# B&R Automation Studio project SuperTrak_Distribution (part 3)

#### ReadErrorMessages.st - Read error messages task
```iecst
(*********************************************************************************
 * Copyright: Bernecker + Rainer
 * Author:  B+R
 * Created:  June 30, 2017/08:15 AM
 *********************************************************************************
 *********************************************************************************
 * Version History:
 * -------------------------------------------------------------------------------
 * V 1.00.0   June 30, 2017/08:15 AM  First Version
 *********************************************************************************
 * Description:
 * -------------------------------------------------------------------------------
 * June 30, 2017/08:15 AM AM V1.00.0:
 * This task is used for Error handling
 * Error number are read from the FUB and converted to messages
 * This messages are used for the visualization
 *********************************************************************************)

ACTION ReadErrorMessages:

	brsmemset(ADR(ErrorInfo),0,SIZEOF(ErrorInfo));

	IF EDGENEG(AcknowledgeAll) THEN
		StControl_0.ErrorReset										:= FALSE;
		FOR Index := 0 TO (SIZEOF(StSection_) / SIZEOF(StSection_[0])) - 1 DO
			StSection_[Index].ErrorReset							:= FALSE;
		END_FOR;
		FOR Index := 0 TO (SIZEOF(StTargetExt_) / SIZEOF(StTargetExt_[0])) - 1 DO
			StTargetExt_[Index].ErrorReset							:= FALSE;
		END_FOR;
		StWritePnu_Region.ErrorReset								:= FALSE;
		StReadPnu_Region.ErrorReset									:= FALSE;
	END_IF;

	FOR Index := 0 TO (SIZEOF(StSection_) / SIZEOF(StSection_[0])) - 1 DO
		////////////////////////////////////////////////////////////
		////////////////////////////////////////////////////////////
		//Check if fault is active to output the correct error msg
		Counter		:= 0;
		FOR FaultBitCounter := 0 TO 31 DO
			IF BIT_TST(StSection_[Index].Info.SuperTrak.SectionFaultBits,FaultBitCounter) THEN
				// Set error
				FaultBit											:= FaultBitCounter;
				ErrorInfo.StSection[Index].ErrorText[Counter]		:= ErrorTexts[FaultBit];
				ErrorInfo.StSection[Index].Error[Counter]			:= FaultBit;
				Counter			:= Counter + 1;
			END_IF;
		END_FOR;

		IF StSection_[Index].StatusID <> stCOM_NO_ERROR THEN
			ErrorInfo.StSection[Index].StatusID				:= StSection_[Index].StatusID;

			// Get the needed text
			CASE ErrorInfo.StSection[Index].StatusID OF
				stCOM_ERR_FB_INSTANCE_REG:
					ErrorInfo.StSection[Index].ErrorText[Counter]:= 'Instance of this function block already registered';

				stCOM_ERR_WRONG_PARAMETER:
					ErrorInfo.StSection[Index].ErrorText[Counter]:= 'Wrong parameter';

				stCOM_ERR_COMMUNICAITON_TIME_OUT:
					ErrorInfo.StSection[Index].ErrorText[Counter]:= 'Timeout for communication to SuperTrak';

				stCOM_ERR_NO_STCONTROL_REG:
					ErrorInfo.StSection[Index].ErrorText[Counter]:= 'There is no instance of StControl registered';

				stCOM_ERR_WRONG_CONFIG:
					ErrorInfo.StSection[Index].ErrorText[Counter]:= 'Address not valid, or Target/Section/PalletID not vaild';

				stCOM_ERR_CMD_NOT_EXECUTED:
					ErrorInfo.StSection[Index].ErrorText[Counter]:= 'Command could not be executed successfully';

				stCOM_ERR_SERVICE_CHANNEL_FAULT:
					ErrorInfo.StSection[Index].ErrorText[Counter]:= 'SuperTrak responded with an error to a service channel request';

				stCOM_ERR_CMD_HANDSHAKE:
					ErrorInfo.StSection[Index].ErrorText[Counter]:= 'CommandComplete flag is true before command execution';

			END_CASE;
		END_IF;

		////////////////////////////////////////////////////////////
		////////////////////////////////////////////////////////////
		//Check if warning is active to output the correct error msg
		Counter		:= 0;
		FOR FaultBitCounter := 0 TO 31 DO
			IF BIT_TST(StSection_[Index].Info.SuperTrak.SectionWarningBits,FaultBitCounter) THEN
				// Set warning
				WarningBit											:= FaultBitCounter;
				ErrorInfo.StSection[Index].WarningText[Counter]		:= WarningTexts[WarningBit];
				ErrorInfo.StSection[Index].Warning[Counter]			:= WarningBit;
				Counter	:= Counter + 1;
			END_IF;
		END_FOR;

		IF StSection_[Index].StatusID <> stCOM_NO_ERROR THEN
			// Get the needed text
			CASE ErrorInfo.StSection[Index].StatusID OF
				stCOM_WRN_ENABLE_SIGNAL_SOURCE:
					ErrorInfo.StSection[Index].WarningText[Counter]:= 'Enable signal source configuration does not allow this command';

				stCOM_INFO_COMM_STRUCT_TOO_BIG:
					ErrorInfo.StSection[Index].WarningText[Counter]:= 'The communication structure is too big';

			END_CASE;
		END_IF;
	END_FOR;

	///////////////////////////////////////////////////////////
	///////////////////////////////////////////////////////////
	// Use the actual selected Section to display
	// Count up the section on the Temperatures Visu page
	IF EDGEPOS(CountUpAlarm) THEN
		VisuAlarmSection		:= VisuAlarmSection + 1;
		// Check for last section
		IF VisuAlarmSection = (MAX_SECTIONS+1) THEN
			VisuAlarmSection	:= 1;
		END_IF;
		CountUpAlarm			:= FALSE;
		// Count down the section on the Temperatures Visu page
	ELSIF EDGEPOS(CountDownAlarm) THEN
		VisuAlarmSection		:= VisuAlarmSection - 1;
		// Check for first section
		IF VisuAlarmSection = 0 THEN
			VisuAlarmSection	:= MAX_SECTIONS;
		END_IF;
		CountDownAlarm			:= FALSE;
	END_IF;

	VisuAlarmSectionText		:= ErrorInfo.StSection[VisuAlarmSection-1].ErrorText;
	VisuWarningSectionText		:= ErrorInfo.StSection[VisuAlarmSection-1].WarningText;

	IF AcknowledgeSelectedSection AND AcknowledgeAll = FALSE THEN
		StSection_[VisuAlarmSection-1].ErrorReset		:= TRUE;
	END_IF;

	///////////////////////////////////////////////////////////
	///////////////////////////////////////////////////////////
	// Check if fault is active to output the correct error msg
	Counter	:= 0;
	FOR Index := 0 TO (SIZEOF(StTargetExt_) / SIZEOF(StTargetExt_[0])) - 1 DO
		// Get the StatusID of the FUB
		IF StTargetExt_[Index].StatusID <> stCOM_NO_ERROR THEN
			ErrorInfo.StTargetExt.StatusID[Counter]			:= StTargetExt_[Index].StatusID;
			ErrorInfo.StTargetExt.TargetID[Counter]			:= Index + 1;

			// Get the needed text
			CASE ErrorInfo.StTargetExt.StatusID[Counter] OF
				stCOM_ERR_FB_INSTANCE_REG:
					ErrorInfo.StTargetExt.ErrorText[Counter]:= 'Instance of this function block already registered';

				stCOM_ERR_WRONG_PARAMETER:
					ErrorInfo.StTargetExt.ErrorText[Counter]:= 'Wrong parameter';

				stCOM_ERR_COMMUNICAITON_TIME_OUT:
					ErrorInfo.StTargetExt.ErrorText[Counter]:= 'Timeout for communication to SuperTrak';

				stCOM_ERR_NO_STCONTROL_REG:
					ErrorInfo.StTargetExt.ErrorText[Counter]:= 'There is no instance of StControl registered';

				stCOM_ERR_WRONG_CONFIG:
					ErrorInfo.StTargetExt.ErrorText[Counter]:= 'Address not valid, or Target/Section/PalletID not vaild';

				stCOM_ERR_CMD_NOT_EXECUTED:
					ErrorInfo.StTargetExt.ErrorText[Counter]:= 'Command could not be executed successfully';

				stCOM_ERR_SERVICE_CHANNEL_FAULT:
					ErrorInfo.StTargetExt.ErrorText[Counter]:= 'SuperTrak responded with an error to a service channel request';

				stCOM_ERR_CMD_HANDSHAKE:
					ErrorInfo.StTargetExt.ErrorText[Counter]:= 'CommandComplete flag is true before command execution';

				stCOM_WRN_ENABLE_SIGNAL_SOURCE:
					ErrorInfo.StTargetExt.ErrorText[Counter]:= 'Enable signal source configuration does not allow this command';

				stCOM_INFO_COMM_STRUCT_TOO_BIG:
					ErrorInfo.StTargetExt.ErrorText[Counter]:= 'The communication structure is too big';

			END_CASE;
			Counter	:= Counter + 1;
		END_IF;
	END_FOR;

	IF AcknowledgeSelectedTarget AND AcknowledgeAll = FALSE THEN
		IF (ErrorInfo.StTargetExt.TargetID[SelectedTarget] -1) >= 0 AND (ErrorInfo.StTargetExt.TargetID[SelectedTarget] -1) < 255 THEN
			StTargetExt_[ErrorInfo.StTargetExt.TargetID[SelectedTarget] -1].ErrorReset		:= TRUE;
		END_IF;
	ELSIF AcknowledgeAll = FALSE THEN
		IF (ErrorInfo.StTargetExt.TargetID[SelectedTarget] -1) >= 0 AND (ErrorInfo.StTargetExt.TargetID[SelectedTarget] -1) < 255 THEN
			StTargetExt_[ErrorInfo.StTargetExt.TargetID[SelectedTarget] -1].ErrorReset		:= FALSE;
		END_IF;
	END_IF;

	///////////////////////////////////////////////////////////
	///////////////////////////////////////////////////////////
	// Check if fault is active to output the correct error msg
	Counter	:= 0;
	FOR Index := 0 TO (SIZEOF(StPallet_) / SIZEOF(StPallet_[0])) - 1 DO
		// Get the StatusID of the FUB
		IF StPallet_[Index].StatusID <> stCOM_NO_ERROR THEN
			ErrorInfo.StPallet.StatusID[Counter]			:= StPallet_[Index].StatusID;
			ErrorInfo.StPallet.ShuttleID[Counter]			:= Index + 1;

			// Get the needed text
			CASE ErrorInfo.StPallet.StatusID[Counter] OF
				stCOM_ERR_FB_INSTANCE_REG:
					ErrorInfo.StPallet.ErrorText[Counter]:= 'Instance of this function block already registered';

				stCOM_ERR_WRONG_PARAMETER:
					ErrorInfo.StPallet.ErrorText[Counter]:= 'Wrong parameter';

				stCOM_ERR_COMMUNICAITON_TIME_OUT:
					ErrorInfo.StPallet.ErrorText[Counter]:= 'Timeout for communication to SuperTrak';

				stCOM_ERR_NO_STCONTROL_REG:
					ErrorInfo.StPallet.ErrorText[Counter]:= 'There is no instance of StControl registered';

				stCOM_ERR_WRONG_CONFIG:
					ErrorInfo.StPallet.ErrorText[Counter]:= 'Address not valid, or Target/Section/PalletID not vaild';

				stCOM_ERR_CMD_NOT_EXECUTED:
					ErrorInfo.StPallet.ErrorText[Counter]:= 'Command could not be executed successfully';

				stCOM_ERR_SERVICE_CHANNEL_FAULT:
					ErrorInfo.StPallet.ErrorText[Counter]:= 'SuperTrak responded with an error to a service channel request';

				stCOM_ERR_CMD_HANDSHAKE:
					ErrorInfo.StPallet.ErrorText[Counter]:= 'CommandComplete flag is true before command execution';

				stCOM_WRN_ENABLE_SIGNAL_SOURCE:
					ErrorInfo.StPallet.ErrorText[Counter]:= 'Enable signal source configuration does not allow this command';

				stCOM_INFO_COMM_STRUCT_TOO_BIG:
					ErrorInfo.StPallet.ErrorText[Counter]:= 'The communication structure is too big';

			END_CASE;
			Counter	:= Counter + 1;
		END_IF;
	END_FOR;

	IF AcknowledgeSelectedShuttle AND AcknowledgeAll = FALSE THEN
		IF (ErrorInfo.StPallet.ShuttleID[SelectedShuttle] -1) >= 0 AND (ErrorInfo.StPallet.ShuttleID[SelectedShuttle] -1) < 255 THEN
			StPallet_[ErrorInfo.StPallet.ShuttleID[SelectedShuttle] -1].ErrorReset		:= TRUE;
		END_IF;
	ELSIF AcknowledgeAll = FALSE THEN
		IF (ErrorInfo.StPallet.ShuttleID[SelectedShuttle] -1) >= 0 AND (ErrorInfo.StPallet.ShuttleID[SelectedShuttle] -1) < 255 THEN
			StPallet_[ErrorInfo.StPallet.ShuttleID[SelectedShuttle] -1].ErrorReset		:= FALSE;
		END_IF;
	END_IF;

	///////////////////////////////////////////////////////////
	///////////////////////////////////////////////////////////
	//Check if fault is active to output the correct error msg
	ErrorInfo.StReadPnu_Region.StatusID			:= StReadPnu_Region.StatusID;
	// Get the needed text
	CASE ErrorInfo.StReadPnu_Region.StatusID OF
		stCOM_ERR_FB_INSTANCE_REG:
			ErrorInfo.StReadPnu_Region.ErrorText:= 'Instance of this function block already registered';

		stCOM_ERR_WRONG_PARAMETER:
			ErrorInfo.StReadPnu_Region.ErrorText:= 'Wrong parameter';

		stCOM_ERR_COMMUNICAITON_TIME_OUT:
			ErrorInfo.StReadPnu_Region.ErrorText:= 'Timeout for communication to SuperTrak';

		stCOM_ERR_NO_STCONTROL_REG:
			ErrorInfo.StReadPnu_Region.ErrorText:= 'There is no instance of StControl registered';

		stCOM_ERR_WRONG_CONFIG:
			ErrorInfo.StReadPnu_Region.ErrorText:= 'Address not valid, or Target/Section/PalletID not vaild';

		stCOM_ERR_CMD_NOT_EXECUTED:
			ErrorInfo.StReadPnu_Region.ErrorText:= 'Command could not be executed successfully';

		stCOM_ERR_SERVICE_CHANNEL_FAULT:
			ErrorInfo.StReadPnu_Region.ErrorText:= 'SuperTrak responded with an error to a service channel request';

		stCOM_ERR_CMD_HANDSHAKE:
			ErrorInfo.StReadPnu_Region.ErrorText:= 'CommandComplete flag is true before command execution';

		stCOM_WRN_ENABLE_SIGNAL_SOURCE:
			ErrorInfo.StReadPnu_Region.ErrorText:= 'Enable signal source configuration does not allow this command';

		stCOM_INFO_COMM_STRUCT_TOO_BIG:
			ErrorInfo.StReadPnu_Region.ErrorText:= 'The communication structure is too big';

	END_CASE;

	///////////////////////////////////////////////////////////
	///////////////////////////////////////////////////////////
	//Check if fault is active to output the correct error msg
	ErrorInfo.StWritePnu_Region.StatusID		:= StWritePnu_Region.StatusID;
	// Get the needed text
	CASE ErrorInfo.StWritePnu_Region.StatusID OF
		stCOM_ERR_FB_INSTANCE_REG:
			ErrorInfo.StWritePnu_Region.ErrorText:= 'Instance of this function block already registered';

		stCOM_ERR_WRONG_PARAMETER:
			ErrorInfo.StWritePnu_Region.ErrorText:= 'Wrong parameter';

		stCOM_ERR_COMMUNICAITON_TIME_OUT:
			ErrorInfo.StWritePnu_Region.ErrorText:= 'Timeout for communication to SuperTrak';

		stCOM_ERR_NO_STCONTROL_REG:
			ErrorInfo.StWritePnu_Region.ErrorText:= 'There is no instance of StControl registered';

		stCOM_ERR_WRONG_CONFIG:
			ErrorInfo.StWritePnu_Region.ErrorText:= 'Address not valid, or Target/Section/PalletID not vaild';

		stCOM_ERR_CMD_NOT_EXECUTED:
			ErrorInfo.StWritePnu_Region.ErrorText:= 'Command could not be executed successfully';

		stCOM_ERR_SERVICE_CHANNEL_FAULT:
			ErrorInfo.StWritePnu_Region.ErrorText:= 'SuperTrak responded with an error to a service channel request';

		stCOM_ERR_CMD_HANDSHAKE:
			ErrorInfo.StWritePnu_Region.ErrorText:= 'CommandComplete flag is true before command execution';

		stCOM_WRN_ENABLE_SIGNAL_SOURCE:
			ErrorInfo.StWritePnu_Region.ErrorText:= 'Enable signal source configuration does not allow this command';

		stCOM_INFO_COMM_STRUCT_TOO_BIG:
			ErrorInfo.StWritePnu_Region.ErrorText:= 'The communication structure is too big';

	END_CASE;

	///////////////////////////////////////////////////////////
	///////////////////////////////////////////////////////////
	//Check if fault is active to output the correct error msg
	Counter		:= 0;
	FOR FaultBitCounter := 0 TO 31 DO
		IF BIT_TST(StControl_0.Info.SuperTrak.SystemFaultBits,FaultBitCounter) THEN
			// Set error
			FaultBit									:= FaultBitCounter;
			ErrorInfo.StControl.Error[Counter]			:= FaultBit;
			ErrorInfo.StControl.ErrorText[Counter]		:= ErrorTexts[FaultBit];
			Counter			:= Counter + 1;
		END_IF;
	END_FOR;

	IF StControl_0.StatusID <> stCOM_NO_ERROR THEN
		ErrorInfo.StControl.StatusID					:= StControl_0.StatusID;

		// Get the needed text
		CASE ErrorInfo.StControl.StatusID OF
			stCOM_ERR_FB_INSTANCE_REG:
				ErrorInfo.StControl.ErrorText[Counter]:= 'Instance of this function block already registered';

			stCOM_ERR_WRONG_PARAMETER:
				ErrorInfo.StControl.ErrorText[Counter]:= 'Wrong parameter';

			stCOM_ERR_COMMUNICAITON_TIME_OUT:
				ErrorInfo.StControl.ErrorText[Counter]:= 'Timeout for communication to SuperTrak';

			stCOM_ERR_NO_STCONTROL_REG:
				ErrorInfo.StControl.ErrorText[Counter]:= 'There is no instance of StControl registered';

			stCOM_ERR_WRONG_CONFIG:
				ErrorInfo.StControl.ErrorText[Counter]:= 'Address not valid, or Target/Section/PalletID not vaild';

			stCOM_ERR_CMD_NOT_EXECUTED:
				ErrorInfo.StControl.ErrorText[Counter]:= 'Command could not be executed successfully';

			stCOM_ERR_SERVICE_CHANNEL_FAULT:
				ErrorInfo.StControl.ErrorText[Counter]:= 'SuperTrak responded with an error to a service channel request';

			stCOM_ERR_CMD_HANDSHAKE:
				ErrorInfo.StControl.ErrorText[Counter]:= 'CommandComplete flag is true before command execution';

		END_CASE;
	END_IF;

	////////////////////////////////////////////////////////////
	////////////////////////////////////////////////////////////
	//Check if warning is active to output the correct error msg
	Counter		:= 0;
	FOR FaultBitCounter := 0 TO 31 DO
		IF BIT_TST(StControl_0.Info.SuperTrak.SystemWarningBits,FaultBitCounter) THEN
			// Set Warning
			WarningBit								:= FaultBitCounter;
			ErrorInfo.StControl.Warning[Counter]	:= WarningBit;
			ErrorInfo.StControl.WarningText[Counter]:= WarningTexts[WarningBit];
			Counter	:= Counter + 1;
		END_IF;
	END_FOR;

	IF StControl_0.StatusID <> stCOM_NO_ERROR THEN
		// Get the needed text
		CASE ErrorInfo.StControl.StatusID OF
			stCOM_WRN_ENABLE_SIGNAL_SOURCE:
				ErrorInfo.StControl.WarningText[Counter]:= 'Enable signal source configuration does not allow this command';

			stCOM_INFO_COMM_STRUCT_TOO_BIG:
				ErrorInfo.StControl.WarningText[Counter]:= 'The communication structure is too big';

		END_CASE;
	END_IF;

	ErrorCode	:= 0;
	////////////////////////////////////////////////////////////
	////////////////////////////////////////////////////////////
	//Check for error in FUB
	ErrorInfo.HmiWriteParID.StatusID			:= HmiWriteParID_0.StatusID;
	// Get the needed text
	CASE ErrorInfo.HmiWriteParID.StatusID OF
		HMI_ERR_FB_INSTANCE_REG:
			ErrorInfo.HmiWriteParID.ErrorText	:= 'Instance of this function block already registered';

		HMI_ERR_WRONG_PARAMETER:
			ErrorInfo.HmiWriteParID.ErrorText	:= 'Wrong parameter';

		HMI_ERR_COMMUNICAITON_TIME_OUT:
			ErrorInfo.HmiWriteParID.ErrorText	:= 'Timeout for communication to SuperTrak';

		HMI_ERR_NO_HMICONTROL_REG:
			ErrorInfo.HmiWriteParID.ErrorText	:= 'There is no instance of HmiControl registered';

		HMI_ERR_WRONG_CONFIG:
			ErrorInfo.HmiWriteParID.ErrorText	:= 'Address not valid, or Target/Section/PalletID not vaild';

		HMI_ERR_CMD_NOT_EXECUTED:
			ErrorInfo.HmiWriteParID.ErrorText:= 'Command could not be executed successfully';
			IF HmiWriteParID_0.Info.ErrorCode <> 0 THEN
				ErrorCode						:= HmiWriteParID_0.Info.ErrorCode;
				brsstrcpy(ADR(ErrorInfo.HmiWriteParID.ErrorText),ADR(HmiErrorTexts[ErrorCode]));
			END_IF;

		HMI_ERR_SERVICE_CHANNEL_FAULT:
			ErrorInfo.HmiWriteParID.ErrorText	:= 'SuperTrak responded with an error to a service channel request';

		HMI_ERR_CMD_HANDSHAKE:
			ErrorInfo.HmiWriteParID.ErrorText	:= 'CommandComplete flag is true before command execution';

		HMI_WRN_ENABLE_SIGNAL_SOURCE:
			ErrorInfo.HmiWriteParID.ErrorText	:= 'Enable signal source configuration does not allow this command';

		HMI_INFO_COMM_STRUCT_TOO_BIG:
			ErrorInfo.HmiWriteParID.ErrorText	:= 'The communication structure is too big';

	END_CASE;

	ErrorCode	:= 0;
	////////////////////////////////////////////////////////////
	////////////////////////////////////////////////////////////
	//Check for error in FUB
	ErrorInfo.HmiReadParID.StatusID				:= HmiReadParID_0.StatusID;
	// Get the needed text
	CASE ErrorInfo.HmiReadParID.StatusID OF
		HMI_ERR_FB_INSTANCE_REG:
			ErrorInfo.HmiReadParID.ErrorText	:= 'Instance of this function block already registered';

		HMI_ERR_WRONG_PARAMETER:
			ErrorInfo.HmiReadParID.ErrorText	:= 'Wrong parameter';

		HMI_ERR_COMMUNICAITON_TIME_OUT:
			ErrorInfo.HmiReadParID.ErrorText	:= 'Timeout for communication to SuperTrak';

		HMI_ERR_NO_HMICONTROL_REG:
			ErrorInfo.HmiReadParID.ErrorText	:= 'There is no instance of HmiControl registered';

		HMI_ERR_WRONG_CONFIG:
			ErrorInfo.HmiReadParID.ErrorText	:= 'Address not valid, or Target/Section/PalletID not vaild';

		HMI_ERR_CMD_NOT_EXECUTED:
			ErrorInfo.HmiReadParID.ErrorText	:= 'Command could not be executed successfully';
			IF HmiReadParID_0.Info.ErrorCode <> 0 THEN
				ErrorCode						:= HmiReadParID_0.Info.ErrorCode;
				brsstrcpy(ADR(ErrorInfo.HmiReadParID.ErrorText),ADR(HmiErrorTexts[ErrorCode]));
			END_IF;

		HMI_ERR_SERVICE_CHANNEL_FAULT:
			ErrorInfo.HmiReadParID.ErrorText	:= 'SuperTrak responded with an error to a service channel request';

		HMI_ERR_CMD_HANDSHAKE:
			ErrorInfo.HmiReadParID.ErrorText	:= 'CommandComplete flag is true before command execution';

		HMI_WRN_ENABLE_SIGNAL_SOURCE:
			ErrorInfo.HmiReadParID.ErrorText	:= 'Enable signal source configuration does not allow this command';

		HMI_INFO_COMM_STRUCT_TOO_BIG:
			ErrorInfo.HmiReadParID.ErrorText	:= 'The communication structure is too big';

	END_CASE;

END_ACTION
```

#### ReadTemp.st - Read temperatures
```iecst
(*********************************************************************************
 * Copyright: Bernecker + Rainer
 * Author:  B+R
 * Created:  June 28, 2017/08:43 AM
 *********************************************************************************
 *********************************************************************************
 * Version History:
 * -------------------------------------------------------------------------------
 * V 1.00.0   June 28, 2017/08:43 AM  First Version
 *********************************************************************************
 * Description:
 * -------------------------------------------------------------------------------
 * June 28, 2017/08:43 AM V1.00.0:
 * This task is reading the temperatures OF a SuperTrak.
 * The variables for the visualization are set
 *********************************************************************************)

ACTION ReadTemp:

	StartIndex	:= 0;
	SuperTrakServChanRead(SectionID,TemperatureID,StartIndex,SIZEOF(Temperatures.Section[SectionID].Value)/SIZEOF(Temperatures.Section[SectionID].Value[0]),ADR(Temperatures.Section[SectionID]),SIZEOF(Temperatures.Section[SectionID]));

	// Read all sensors which are enabled or disabled by the user
	SuperTrakServChanRead(SectionID,1170,StartIndex,1, ADR(Temperatures.Section[SectionID].DefaultMask), SIZEOF(Temperatures.Section[SectionID].DefaultMask));
	SuperTrakServChanRead(SectionID,1169,StartIndex,1, ADR(Temperatures.Section[SectionID].UserEnableMask), SIZEOF(Temperatures.Section[SectionID].UserEnableMask));
	SuperTrakServChanRead(SectionID,1168,StartIndex,1, ADR(Temperatures.Section[SectionID].UserDisableMask), SIZEOF(Temperatures.Section[SectionID].UserDisableMask));

	// Calculate effective mask for temperature sensors
	Temperatures.Section[SectionID].EffectiveMask := Temperatures.Section[SectionID].UserEnableMask OR(Temperatures.Section[SectionID].DefaultMask AND NOT(Temperatures.Section[SectionID].UserDisableMask));

	// Mapping of active temperature sensors
	Temperatures.Section[SectionID].SensorActivated[0] := Temperatures.Section[SectionID].EffectiveMask.0;
	Temperatures.Section[SectionID].SensorActivated[1] := Temperatures.Section[SectionID].EffectiveMask.1;
	Temperatures.Section[SectionID].SensorActivated[2] := Temperatures.Section[SectionID].EffectiveMask.2;
	Temperatures.Section[SectionID].SensorActivated[3] := Temperatures.Section[SectionID].EffectiveMask.3;
	Temperatures.Section[SectionID].SensorActivated[4] := Temperatures.Section[SectionID].EffectiveMask.4;
	Temperatures.Section[SectionID].SensorActivated[5] := Temperatures.Section[SectionID].EffectiveMask.5;
	Temperatures.Section[SectionID].SensorActivated[6] := Temperatures.Section[SectionID].EffectiveMask.6;

	Temperatures.Section[SectionID].SensorActivated[8] := Temperatures.Section[SectionID].EffectiveMask.8;
	Temperatures.Section[SectionID].SensorActivated[9] := Temperatures.Section[SectionID].EffectiveMask.9;
	Temperatures.Section[SectionID].SensorActivated[10] := Temperatures.Section[SectionID].EffectiveMask.10;
	Temperatures.Section[SectionID].SensorActivated[11] := Temperatures.Section[SectionID].EffectiveMask.11;
	Temperatures.Section[SectionID].SensorActivated[12] := Temperatures.Section[SectionID].EffectiveMask.12;
	Temperatures.Section[SectionID].SensorActivated[13] := Temperatures.Section[SectionID].EffectiveMask.13;
	Temperatures.Section[SectionID].SensorActivated[14] := Temperatures.Section[SectionID].EffectiveMask.14;

	// Search for error/warning
	// To get the temperature --> /100
	FOR StartIndex := 0 TO 15 DO
		IF Temperatures.Section[VisuSection].SensorActivated[StartIndex] THEN
				Temperatures.Section[VisuSection].Warning[StartIndex]	:= (UINT_TO_REAL(Temperatures.Section[VisuSection].Value[StartIndex])/100) > WarningTemperature;
				Temperatures.Section[VisuSection].Error[StartIndex]	:= (UINT_TO_REAL(Temperatures.Section[VisuSection].Value[StartIndex])/100) > ErrorTemperature;
		END_IF
	END_FOR;

	IF SectionID = CONFIG_ST_MAX_SECTIONS THEN
		SectionID					:= 1;
	ELSE
		SectionID					:= SectionID+1;
	END_IF;

	// Count up the section on the Temperatures Visu page
	IF EDGEPOS(CountUp) THEN
		VisuSection		:= VisuSection + 1;
		// Check for last section
		IF VisuSection = (MAX_SECTIONS+1) THEN
			VisuSection	:= 1;
		END_IF;
		CountUp			:= FALSE;
		// Count down the section on the Temperatures Visu page
	ELSIF EDGEPOS(CountDown) THEN
		VisuSection		:= VisuSection - 1;
		// Check for first section
		IF VisuSection = 0 THEN
			VisuSection	:= MAX_SECTIONS;
		END_IF;
		CountDown		:= FALSE;
	END_IF;

	// Get the needed section data
	FOR i:= 0 TO 15 DO
		IF Temperatures.Section[VisuSection].SensorActivated[i] THEN
			VisuTemp.Value[i]				:= UINT_TO_REAL(Temperatures.Section[VisuSection].Value[i])/100;
		ELSE
			VisuTemp.Value[i] 				:= 0;
		END_IF
	END_FOR;
	VisuTemp.Error		:= Temperatures.Section[VisuSection].Error;
	VisuTemp.Warning	:= Temperatures.Section[VisuSection].Warning;
END_ACTION
```

#### SetPalletIDs.st - Set pallet IDs
```iecst
(*********************************************************************************
 * Copyright: Bernecker + Rainer
 * Author:  B+R
 * Created:  November 20, 2017/08:15 AM
 *********************************************************************************
 *********************************************************************************
 * Version History:
 * -------------------------------------------------------------------------------
 * V 1.00.0   November 20, 2017/08:15 AM  First Version
 *********************************************************************************
 * Description:
 * -------------------------------------------------------------------------------
 * This task is used for setting Shuttle(Pallet) IDs
 *********************************************************************************)

ACTION SetPalletIDs:

	// Check if actual shuttles has an ID
	IF StTargetExt_[StartTarget-1].PalletPresent AND StTargetExt_[StartTarget-1].PalletID = 0 THEN
		StTargetExt_[StartTarget-1].SetPalletID	:= TRUE;
	// Release the shuttle to a Wait target
	ELSIF StTargetExt_[StartTarget-1].CommandDone AND StTargetExt_[StartTarget-1].SetPalletID THEN
		StTargetExt_[StartTarget-1].SetPalletID	:= FALSE;
		PalletControlParameters[TargetControlParameters[StartTarget-1].PalletConfig.ID-1].AdvancedReleaseConfig.Direction			:= stCOM_DIR_RIGHT;
		PalletControlParameters[TargetControlParameters[StartTarget-1].PalletConfig.ID-1].AdvancedReleaseConfig.DestinationTarget	:= WaitTarget;
		StPallet_[TargetControlParameters[StartTarget-1].PalletConfig.ID-1].ReleaseToTarget											:= TRUE;
		TargetControlParameters[StartTarget-1].PalletConfig.ID	:= TargetControlParameters[StartTarget-1].PalletConfig.ID + 1;
	END_IF;

	// Count the shuttles on the Wait target (Target 2)
	FOR IndexSetIDs := 0 TO (SIZEOF(StPallet_) / SIZEOF(StPallet_[0])) - 1 DO
		IF StPallet_[IndexSetIDs].CommandDone THEN
			StPallet_[IndexSetIDs].ReleaseToTarget	:= FALSE;
		END_IF;
	END_FOR;

	// Release shuttles from Wait target
	IF StTargetExt_[WaitTarget-1].PalletPresent AND NOT(StTargetExt_[WaitTarget-1].ReleaseToTarget) THEN
		TargetControlParameters[WaitTarget-1].AdvancedReleaseConfig.DestinationTarget	:= StartTarget;
		TargetControlParameters[WaitTarget-1].AdvancedReleaseConfig.Direction			:= stCOM_DIR_RIGHT;
		StTargetExt_[WaitTarget-1].ReleaseToTarget	:= TRUE;
		ReleasedShuttles							:= ReleasedShuttles + 1;
	ELSIF StTargetExt_[WaitTarget-1].CommandDone THEN
		StTargetExt_[WaitTarget-1].ReleaseToTarget	:= FALSE;
	END_IF;

	// Check if all shuttles have IDs and are released from Wait target
	IF StTargetExt_[StartTarget-1].PalletPresent AND StTargetExt_[StartTarget-1].PalletID >= 1 AND TargetControlParameters[StartTarget-1].PalletConfig.ID > NumberOfShuttles AND
		ReleasedShuttles = NumberOfShuttles THEN
		IDSet	:= TRUE;
	// Check if all shuttles have an ID. Release shuttles if not all have an ID and wait for the problematic shuttle
	ELSIF StTargetExt_[StartTarget-1].PalletPresent AND StTargetExt_[StartTarget-1].PalletID <> 0 AND TargetControlParameters[StartTarget-1].PalletConfig.ID <= NumberOfShuttles THEN
		StPallet_[StTargetExt_[StartTarget-1].PalletID-1].ReleaseToTarget	:= TRUE;
	END_IF;

END_ACTION
```

#### CheckStandstill.st - Check shuttles for standstill
```iecst
(*********************************************************************************
 * Copyright: Bernecker + Rainer
 * Author:  B+R
 * Created:  November 22, 2017/3:15 PM
 *********************************************************************************
 *********************************************************************************
 * Version History:
 * -------------------------------------------------------------------------------
 * V 1.00.0   November 22, 2017/3:15 PM  First Version
 *********************************************************************************
 * Description:
 * -------------------------------------------------------------------------------
 * November 22, 2017/3:15 PM V1.00.0:
 * This task is used for checking if all shuttles are not moving
 *********************************************************************************)
ACTION CheckStandstill:

	// Check if the shuttle is in standstill
	ShuttlesStandstill	:= TRUE;
	FOR Index := 0 TO (SIZEOF(StPallet_) / SIZEOF(StPallet_[0])) - 1 DO
		PositionDelta[Index].Position		:= ShuttleInfo[Index].position - PositionDelta[Index].PositionOld;
		PositionDelta[Index].PositionOld	:= ShuttleInfo[Index].position;

		IF ABS(PositionDelta[Index].Position) > PositionOffset OR StTargetExt_[WaitTarget-1].PalletPresent THEN
			ShuttlesStandstill	:= FALSE;
		END_IF;

	END_FOR;

END_ACTION
```

#### DisableRegion.st - Disable the region
```iecst
(*********************************************************************************
 * Copyright: Bernecker + Rainer
 * Author:  B+R
 * Created:  November 23, 2017/2:00 PM
 *********************************************************************************
 *********************************************************************************
 * Version History:
 * -------------------------------------------------------------------------------
 * V 1.00.0   November 23, 2017/2:00 PM  First Version
 *********************************************************************************
 * Description:
 * -------------------------------------------------------------------------------
 * November 23, 2017/2:00 PM V1.00.0:
 * This task is used FOR disable the safety region
 *********************************************************************************)

ACTION DisableRegion:
	StWritePnu_Region.Enable			:= TRUE;
	StWritePnu_Region.DataAddress		:= ADR(Region);
	StWritePnu_Region.DataSize			:= SIZEOF(Region);
	StWritePnuPar_Region.ParameterNumber:= 1600;
	StWritePnuPar_Region.ValidDataSize	:= SIZEOF(Region);

	StWritePnu_Region.Write				:= TRUE;

	StReadPnu_Region.Enable				:= TRUE;

	IF StReadPnu_Region.Read = FALSE AND StReadPnu_Region.CommandDone = FALSE AND StReadPnu_Region.Active THEN
		StReadPnu_Region.Read			:= TRUE;
	ELSE
		StReadPnu_Region.Read			:= FALSE;
	END_IF;

	IF StWritePnu_Region.CommandDone AND RegionStatus = 0 THEN
		//Save region configuration
		IF SuperTrakServChanWrite(0,Save_Parameter,0,1,ADR(SaveValue),SIZEOF(SaveValue)) = 0 AND StControl_0.Info.SuperTrak.SystemWarningActive = FALSE THEN
			StWritePnu_Region.Write		:= FALSE;
			RegionDisabled				:= TRUE;
			RegionEnabled				:= FALSE;
			StReadPnu_Region.Enable		:= FALSE;
			StWritePnu_Region.Enable	:= FALSE;
		END_IF;
	END_IF;
END_ACTION
```

#### EnableRegion.st - Enable the region
```iecst
(*********************************************************************************
 * Copyright: Bernecker + Rainer
 * Author:  B+R
 * Created:  November 23, 2017/1:30 PM
 *********************************************************************************
 *********************************************************************************
 * Version History:
 * -------------------------------------------------------------------------------
 * V 1.00.0   November 23, 2017/1:30 PM  First Version
 *********************************************************************************
 * Description:
 * -------------------------------------------------------------------------------
 * November 23, 2017/1:30 PM V1.00.0:
 * This task is used FOR enable the safety region
 *********************************************************************************)

ACTION EnableRegion:
	StWritePnu_Region.Enable				:= TRUE;
	StWritePnu_Region.DataAddress			:= ADR(RegionEnable);
	StWritePnu_Region.DataSize				:= SIZEOF(RegionEnable);
	StWritePnuPar_Region.ParameterNumber	:= 1600;
	StWritePnuPar_Region.ValidDataSize		:= SIZEOF(RegionEnable);

	StWritePnu_Region.Write					:= TRUE;

	IF StWritePnu_Region.Write THEN
		TimerRegionEnable.IN				:= TRUE;
	END_IF;

	IF TimerRegionEnable.Q THEN
		TimerRegionEnable.IN				:= FALSE;
		StWritePnu_Region.Write				:= FALSE;
	END_IF;

	StReadPnu_Region.Enable					:= TRUE;
	StReadPnu_Region.DataAddress			:= ADR(RegionStatus);
	StReadPnu_Region.DataSize				:= SIZEOF(RegionStatus);
	StReadPnuPar_Region.ParameterNumber		:= 1600;
	StReadPnuPar_Region.StartParameterIndex	:= 0;

	IF StReadPnu_Region.Read = FALSE AND StReadPnu_Region.CommandDone = FALSE THEN
		StReadPnu_Region.Read				:= TRUE;
	ELSE
		StReadPnu_Region.Read				:= FALSE;
	END_IF;

	IF StWritePnu_Region.CommandDone AND RegionStatus = 7 THEN
		//Save region configuration
		IF SuperTrakServChanWrite(0,Save_Parameter,0,1,ADR(SaveValue),SIZEOF(SaveValue)) = 0 AND StControl_0.Info.SuperTrak.SystemWarningActive = FALSE THEN
			StWritePnu_Region.Write			:= FALSE;
			RegionEnabled					:= TRUE;
			TimerRegionEnable.IN			:= FALSE;
			StReadPnu_Region.Enable			:= FALSE;
		END_IF;
	END_IF;
END_ACTION
```

#### AlarmX.st - Error Handling with mapp AlarmX
```iecst
(*********************************************************************************
 * Copyright: Bernecker+Rainer
 * Author:    B&R
 * Created:   May 9, 21718/11:27 AM
 *********************************************************************************
 *********************************************************************************
 * Version History:
 * -------------------------------------------------------------------------------
 * V 1.1717.17   May 9, 21718/11:27 AM  First Version
 *********************************************************************************
 * Description:
 * *Contains source code for mappAlarmX
 * *Alarms can be modified in Configuration View under mappServices in Config.mpAlarmXCore
 *********************************************************************************)

ACTION AlarmX:

	// read Service Channel of each Section with StSection to identifey errors and warnings
	FOR Index := 0 TO (SIZEOF(StSection_) / SIZEOF(StSection_[0])) - 1 DO
		(* Errors & Warnings on each bit*)
		FOR counter := 0 TO 31 DO
			// Errors
			IF BIT_TST(StSection_[Index].Info.SuperTrak.SectionFaultBits,counter) THEN
				IF MpAlarmXCheckState(gAlarmXCore, ErrorStrings[counter],mpALARMX_STATE_NONE) THEN
					MpAlarmXSet(gAlarmXCore, ErrorStrings[counter]);
					ErrorBitOnSection[Index].ErrorBitSet[counter]	:= TRUE;
				END_IF;
			ELSE
				ErrorBitOnSection[Index].ErrorBitSet[counter]	:= FALSE;
			END_IF;

			ReadyToReset	:= TRUE;
			FOR Index2 := 0 TO (SIZEOF(StSection_) / SIZEOF(StSection_[0])) - 1 DO
				IF ErrorBitOnSection[Index2].ErrorBitSet[counter] THEN
					ReadyToReset	:= FALSE;
				END_IF;
			END_FOR;

			IF NOT BIT_TST(StSection_[Index].Info.SuperTrak.SectionFaultBits,counter) AND ReadyToReset THEN
				MpAlarmXReset(gAlarmXCore, ErrorStrings[counter]);
			END_IF;
			//Warnings
			IF BIT_TST(StSection_[Index].Info.SuperTrak.SectionWarningBits,counter) AND NOT WarningBitSection[Index].ErrorBitSet[counter] THEN
				IF MpAlarmXCheckState(gAlarmXCore, WarningStrings[counter],mpALARMX_STATE_NONE) THEN
					MpAlarmXSet(gAlarmXCore, WarningStrings[counter]);
					WarningBitSection[Index].ErrorBitSet[counter] := TRUE;
				END_IF;
			ELSE
				WarningBitSection[Index].ErrorBitSet[counter] := FALSE;
			END_IF;

			ReadyToReset	:= TRUE;
			FOR Index2 := 0 TO (SIZEOF(StSection_) / SIZEOF(StSection_[0])) - 1 DO
				IF WarningBitSection[Index].ErrorBitSet[counter] THEN
					ReadyToReset	:= FALSE;
				END_IF;
			END_FOR;

			IF BIT_TST(StSection_[Index].Info.SuperTrak.SectionWarningBits,counter) AND ReadyToReset THEN
					MpAlarmXReset(gAlarmXCore, WarningStrings[counter]);

			END_IF;
		END_FOR;
	END_FOR;

	/////////////////////////////////////////////////////////////////////////////////////////////////////////////////////////////////////////////////////////
	/////////////////////////////////////////////////////////////////////////////////////////////////////////////////////////////////////////////////////////
	(* Errors & Warnings on each bit*)
	FOR counter := 0 TO 31 DO
		// Errors
		IF BIT_TST(StControl_0.Info.SuperTrak.SystemFaultBits,counter) THEN
			IF MpAlarmXCheckState(gAlarmXCore, ErrorStrings1[counter],mpALARMX_STATE_NONE) THEN
				MpAlarmXSet(gAlarmXCore, ErrorStrings1[counter]);
			END_IF;
		END_IF;

		IF NOT BIT_TST(StControl_0.Info.SuperTrak.SystemFaultBits,counter) THEN
			MpAlarmXReset(gAlarmXCore, ErrorStrings1[counter]);
		END_IF;

		//Warnings
		IF BIT_TST(StControl_0.Info.SuperTrak.SystemWarningBits,counter) THEN
			IF MpAlarmXCheckState(gAlarmXCore, WarningStrings1[counter],mpALARMX_STATE_NONE) THEN
				MpAlarmXSet(gAlarmXCore, WarningStrings1[counter]);
			END_IF;
		END_IF;
		IF BIT_TST(StControl_0.Info.SuperTrak.SystemWarningBits,counter) THEN
			MpAlarmXReset(gAlarmXCore, WarningStrings1[counter]);

		END_IF;

	END_FOR;

	/////////////////////////////////////////////////////////////////////////////////////////////////////////////////////////////////////////////////////////
	/////////////////////////////////////////////////////////////////////////////////////////////////////////////////////////////////////////////////////////
	IF SaveHistory AND NOT MpAlarmXHistory_0.CommandBusy THEN
		MpAlarmXHistory_0.Export := TRUE;
	END_IF;

	IF MpAlarmXHistory_0.CommandDone THEN
		SaveHistory := FALSE;
		MpAlarmXHistory_0.Export := FALSE;
	END_IF;

	(* Function block calls *)
	MpAlarmXCore_0();
	MpAlarmXHistory_0();

END_ACTION
```

#### AlarmXInit.st - Init Function blocks for mapp AlarmX
```iecst
(*********************************************************************************
 * Copyright: Bernecker+Rainer
 * Author:    B&R
 * Created:   May 9, 2018/11:27 AM
 *********************************************************************************
 *********************************************************************************
 * Version History:
 * -------------------------------------------------------------------------------
 * V 1.00.0   May 9, 2018/11:27 AM  First Version
 *********************************************************************************
 * Description:
 * *Contains function block init parameters
 * *Alarms can be modified in Configuration View under mappServices in Config.mpAlarmXCore
 *********************************************************************************)

ACTION AlarmXInit:
		(* Setting up mpAlarmX Parameters *)
	MpAlarmXCore_0.MpLink := ADR(gAlarmXCore);
	MpAlarmXCore_0.Enable := TRUE;

	(* Setting parameter for mpAlarmXHistory *)
	MpAlarmXHistory_0.MpLink := ADR(gAlarmXHistory);
	MpAlarmXHistory_0.Enable := TRUE;
	IF DiagCpuIsSimulated() THEN
		MpAlarmXHistory_0.DeviceName := ADR('Sim');
	ELSE
		MpAlarmXHistory_0.DeviceName := ADR('CFast');
	END_IF;
END_ACTION
```

#### InitParID.st
```iecst
(*********************************************************************************
 * Copyright: Bernecker+Rainer
 * Author:    B&R
 * Created:   June 12, 2018/13:10 AM
 *********************************************************************************
 *********************************************************************************
 * Version History:
 * -------------------------------------------------------------------------------
 * V 1.00.0   June 12, 2018/13:10 AM  First Version
 *********************************************************************************
 * Description:
 * *Contains function block init parameters
 *********************************************************************************)

ACTION InitParID:

	HmiControl_0.HMILink			:= ADR(HmiLink);
	HmiControl_0.Enable				:= TRUE;

	HmiWriteParID_0.HMILink			:= ADR(HmiLink);
	HmiWriteParID_0.Parameters		:= ADR(HmiWritePar);

	HmiReadParID_0.HMILink			:= ADR(HmiLink);
	HmiReadParID_0.Parameters		:= ADR(HmiReadPar);

	HmiWritePar.ParameterValueCount	:= 1;
	HmiReadPar.ParameterValueCount	:= 1;

END_ACTION
```

#### ShuttleConfig.st
```iecst
ACTION ShuttleConfig:

	///////////////////////////////////////////////////////////
	///////////////////////////////////////////////////////////
	// Use the actual selected shuttle to display
	// Count up the shuttle on the Temperatures Visu page
	IF EDGEPOS(CountUpShuttle) THEN
		VisuShuttle				:= VisuShuttle + 1;
		// Check for last section
		IF VisuShuttle = (StControl_0.Info.SuperTrak.NrOfPallets+1) THEN
			VisuShuttle			:= 1;
		END_IF;
		CountUpShuttle			:= FALSE;

		Config_ShelfWidth				:= PalletControlParameters[VisuShuttle-1].PalletConfig.Shelf.ShelfWidth;
		Config_OffsetFromCenter			:= PalletControlParameters[VisuShuttle-1].PalletConfig.Shelf.OffsetFromCenter;
		Config_ControlGainSetIndex		:= PalletControlParameters[VisuShuttle-1].PalletConfig.Controller.ControlGainSetIdx;
		Config_FilterWeightMoving		:= PalletControlParameters[VisuShuttle-1].PalletConfig.Controller.FilterWeightMoving;
		Config_FilterWeightStationary	:= PalletControlParameters[VisuShuttle-1].PalletConfig.Controller.FilterWeightStationary;

		// Count down the section on the Temperatures Visu page
	ELSIF EDGEPOS(CountDownShuttle) THEN
		VisuShuttle				:= VisuShuttle - 1;
		// Check for first section
		IF VisuShuttle = 0 THEN
			VisuShuttle			:= StControl_0.Info.SuperTrak.NrOfPallets;
		END_IF;
		CountDownShuttle		:= FALSE;

		Config_ShelfWidth				:= PalletControlParameters[VisuShuttle-1].PalletConfig.Shelf.ShelfWidth;
		Config_OffsetFromCenter			:= PalletControlParameters[VisuShuttle-1].PalletConfig.Shelf.OffsetFromCenter;
		Config_ControlGainSetIndex		:= PalletControlParameters[VisuShuttle-1].PalletConfig.Controller.ControlGainSetIdx;
		Config_FilterWeightMoving		:= PalletControlParameters[VisuShuttle-1].PalletConfig.Controller.FilterWeightMoving;
		Config_FilterWeightStationary	:= PalletControlParameters[VisuShuttle-1].PalletConfig.Controller.FilterWeightStationary;
	END_IF;

	PalletControlParameters[VisuShuttle-1].PalletConfig.Shelf.ShelfWidth					:= Config_ShelfWidth;
	PalletControlParameters[VisuShuttle-1].PalletConfig.Shelf.OffsetFromCenter				:= Config_OffsetFromCenter;
	PalletControlParameters[VisuShuttle-1].PalletConfig.Controller.ControlGainSetIdx		:= Config_ControlGainSetIndex;
	PalletControlParameters[VisuShuttle-1].PalletConfig.Controller.FilterWeightMoving		:= Config_FilterWeightMoving;
	PalletControlParameters[VisuShuttle-1].PalletConfig.Controller.FilterWeightStationary	:= Config_FilterWeightStationary;

	StPallet_[VisuShuttle-1].SetPalletShelf				:= Config_SetPalletShelf AND NOT(StPallet_[VisuShuttle-1].SetPalletGain);
	StPallet_[VisuShuttle-1].SetPalletGain				:= Config_SetGain AND NOT(StPallet_[VisuShuttle-1].SetPalletShelf);

	IF StPallet_[VisuShuttle-1].CommandDone THEN
		StPallet_[VisuShuttle-1].SetPalletShelf			:= FALSE;
		StPallet_[VisuShuttle-1].SetPalletGain			:= FALSE;
		Config_SetPalletShelf							:= FALSE;
		Config_SetGain									:= FALSE;
	END_IF;

END_ACTION
```

### Program Logical/Source/SuperTrak/ST_Main (IEC) - Create the Service-Channel to the SuperTrak controller

#### Main.st - Init, cyclic, exit code
```iecst
(*********************************************************************************
 * Copyright: ATS Automation Tooling Systems, Inc. 2015
 *     All rights reserved.
 *********************************************************************************
 *********************************************************************************
 * Description:
 * -------------------------------------------------------------------------------
 * This task configures the internal communication structure AND controlls
 * the SuperTrak system.
 *********************************************************************************)

PROGRAM _INIT
// SuperTrak initialization
	IF DiagCpuIsARsim() THEN
		(* This path can be customized as needed *)
		StoragePath := '/DEVICE=C:\Temp\SuperTrakUser';
	ELSE
		(* CFast card USER partition *)
		StoragePath := '/DEVICE=F:\';
	END_IF;

	// SuperTrak Init function call
	SuperTrakInit(StoragePath, ARSimIPAddress, EthernetInterfaces);

	// Service Channel initialization
	ServiceChannelData.channelId    		:= 1;
	ServiceChannelData.pRequestHeader		:= ADR(gStServiceChannelReqData);
	ServiceChannelData.pResponseHeader		:= ADR(gStServiceChannelResData);
	ServiceChannelData.pRequestValues     	:= ADR(gStServiceChannelReqData) + SIZEOF(ServiceChannelHeader_t);
	ServiceChannelData.pResponseValues    	:= ADR(gStServiceChannelResData) + SIZEOF(ServiceChannelHeader_t);
	ServiceChannelData.requestBufferSize  	:= SIZEOF(gStServiceChannelReqData);
	ServiceChannelData.responseBufferSize  	:= SIZEOF(gStServiceChannelResData);
	ServiceChannelData.state     			:= scSTATE_RECV;

	pResView ACCESS ADR(gStServiceChannelResData);
	pReqView ACCESS ADR(gStServiceChannelReqData);

	// Command interface mapping
	SuperTrakControlInterface[0].pControl  	:= ADR(gStCyclicControlData);
	SuperTrakControlInterface[0].pStatus   	:= ADR(gStCyclicStatusData);
	SuperTrakControlInterface[0].controlSize:= SIZEOF(gStCyclicControlData);
	SuperTrakControlInterface[0].statusSize := SIZEOF(gStCyclicStatusData);

	(* De-configure any "Allow Section Enable" inputs *)
	(* Parameter 1092: Parameter Array Length (UDINT) *)
	(* Parameter 1200: Digital Input Function (UINT) *)
	status := SuperTrakServChanRead(0, 1092, 1200 - 1024, 1, ADR(udintValue), SIZEOF(udintValue));

	IF (status = scERR_SUCCESS) THEN
		count := MIN(UDINT_TO_UINT(udintValue),
		SIZEOF(digitalInputFunction) / SIZEOF(digitalInputFunction[0]));

		status := SuperTrakServChanRead(0, 1200, 0, count, ADR(digitalInputFunction), SIZEOF(digitalInputFunction));

		IF (status = scERR_SUCCESS) THEN
			FOR i := 0 TO count - 1 DO
				(* Input Function 25: Allow Section Enable *)
				IF (digitalInputFunction[i] = 25) THEN
					(* Input Function 0: Not Configured *)
					digitalInputFunction[i] := 0;
					status := SuperTrakServChanWrite(0, 1200, i, 1, ADR(digitalInputFunction[i]), SIZEOF(digitalInputFunction[i]));
				END_IF;
			END_FOR;
		END_IF;
	END_IF;

	(* Ensure that control interface revision 0 is selected *)
	(* Parameter 1444: Control Interface Revision (UINT) *)
	status := SuperTrakServChanRead(0, 1444, 0, 1, ADR(uintValue), SIZEOF(uintValue));

	IF (status = scERR_SUCCESS) THEN
		IF (uintValue <> 0) THEN
			uintValue := 0;
			status := SuperTrakServChanWrite(0, 1444, 0, 1, ADR(uintValue), SIZEOF(uintValue));
		END_IF;
	END_IF;

END_PROGRAM

PROGRAM _CYCLIC

	// Map internal communication structure
	FOR i := 0 TO stMAX_CONTROL_IF_INDEX DO
		SuperTrakProcessControl(i, SuperTrakControlInterface[i]);
	END_FOR;

	// Cylcic SuperTrak control
	SuperTrakCyclic1();

	(* PLC interfaces status *)
	FOR i := 0 TO stMAX_CONTROL_IF_INDEX DO
		SuperTrakProcessStatus(i, SuperTrakControlInterface[i]);
	END_FOR;

	// Service channel handling
	IF ServiceChannelData.state = scSTATE_RECV AND
		pReqView.sequence <> pResView.sequence THEN
		ServiceChannelData.requestSequence  := pReqView.sequence;
		ServiceChannelData.state    		:= scSTATE_EXEC;
	ELSIF ServiceChannelData.state = scSTATE_EXEC OR ServiceChannelData.state = scSTATE_WAIT THEN
		SuperTrakServiceChannel(ServiceChannelData);
	ELSIF ServiceChannelData.state = scSTATE_SEND THEN
		ServiceChannelData.state    		:= scSTATE_RECV;
	END_IF;

END_PROGRAM

PROGRAM _EXIT

 // Clear internal memory
	SuperTrakExit();

END_PROGRAM
```

#### Variables.var - Local variables
```iecst
(********************************************************************
 * Copyright ATS Automation Tooling Systems, Inc. 2015
 * All rights reserved.
 ********************************************************************
 * Local variables
 ********************************************************************)
(*ServiceChannel Handling*)
VAR
	SuperTrakControlInterface : ARRAY[0..stMAX_CONTROL_IF_INDEX] OF SuperTrakControlInterface_t := [stMAX_CONTROL_IF_COUNT((0))];
	ServiceChannelData : ServiceChannel_t := (0);
	pResView : REFERENCE TO ServiceChannelHeader_t;
	pReqView : REFERENCE TO ServiceChannelHeader_t;
END_VAR
(*SuperTrak Init Parameters*)
VAR
	ARSimIPAddress : STRING[15] := '127.0.0.1'; (*IP Adress of the ArSim*)
	EthernetInterfaces : STRING[31] := 'IF3,IF4'; (*Existing Ethernet Interfaces on APC*)
	StoragePath : STRING[127];
END_VAR
(*Insert your comment here.*)
VAR
	i : UINT := 0;
	status : UINT := 0;
	count : UINT := 0;
	digitalInputFunction : ARRAY[0..7] OF UINT := [8(0)];
	udintValue : UDINT;
	uintValue : UINT;
END_VAR
```

### Program Logical/Source/SuperTrak/ST_Visu (IEC) - Connection to Scene Viewer

#### Cyclic.st - Cyclic code
```iecst
(*********************************************************************************
 * Copyright Bernecker + Rainer 2015
 * Copyright ATS Automation Tooling Systems, Inc. 2017-2018
 * All rights reserved.
 * -------------------------------------------------------------------------------
 * This task calculates the actual pallet positions in the room based on the
 * section number and the position of the pallet in the section.
 * It is also hiding unused sections and/or pallets.
 * This data is then provided to B&R Scene Viewer.
 *********************************************************************************)

PROGRAM _INIT

	visuStep := 0;

END_PROGRAM

PROGRAM _CYCLIC

	CASE visuStep OF
		visuSTEP_INITIALIZE:
			visuStep := visuSTEP_GET_SECTION_COUNT;

		visuSTEP_GET_SECTION_COUNT:
			// read parameter 1080: section count
			result := SuperTrakServChanRead(0, 1080, 0, 1, ADR(sectionCount), SIZEOF(sectionCount));

			IF (result = scERR_SUCCESS) AND (sectionCount > 0) THEN
				visuStep := visuSTEP_GET_SECTION_ADDRS;
			ELSE
				visuStep := visuSTEP_ERROR;
			END_IF;

		visuSTEP_GET_SECTION_ADDRS:
			// read parameter 1081: section user address
			result := SuperTrakServChanRead(0, 1081, 0, sectionCount, ADR(servChanResponseUINT), SIZEOF(servChanResponseUINT));

			IF (result = scERR_SUCCESS) THEN
				FOR i := 0 TO sectionCount - 1 DO
					Section[i].userAddress := servChanResponseUINT[i];

					IF (Section[i].userAddress > 0) AND (Section[i].userAddress < 99) THEN
						sectionLookup[ Section[i].userAddress ] := i;
					END_IF;
				END_FOR;

				visuStep := visuSTEP_GET_SECTION_TYPES;
				i := 0;
			ELSE
				visuStep := visuSTEP_ERROR;
			END_IF;

		visuSTEP_GET_SECTION_TYPES:
			// read parameter 1082: section type
			result := SuperTrakServChanRead(UINT_TO_USINT(Section[i].userAddress), 1082, 0, 1, ADR(Section[i].sectionType), SIZEOF(UINT));

			IF (result = scERR_SUCCESS) THEN
				i := i + 1;

				IF (i >= sectionCount) THEN
					visuStep := visuSTEP_SETUP_SECTIONS;
				END_IF;
			ELSE
				visuStep := visuSTEP_ERROR;
			END_IF;

		visuSTEP_SETUP_SECTIONS:
			// Assign visualization models to sections.
			// Mostly assume that the layout is sensible.
			side := 0;
			sideLength[0] := 0;
			sideLength[1] := 0;
			position := 0;
			modelIndex := 0;

			FOR i := 0 TO sectionCount - 1 DO
				Section[i].side := -1;
				Section[i].modelIndex := -1;

				IF (Section[i].sectionType = SECTION_TYPE_1M) OR (Section[i].sectionType = SECTION_TYPE_1M_LP) THEN
					// Straight section models are indexed 0-31 (front) and 32-63 (back).
					IF (side < 2)
						AND (modelIndex >= (side * 32))
						AND (modelIndex < ((side + 1) * 32)) THEN

						Section[i].side := side;
						sideLength[side] := sideLength[side] + 1;

						Data.StraightSectionVisible[modelIndex] := TRUE;
						Section[i].modelIndex := modelIndex;
						modelIndex := modelIndex + 1;

						Section[i].positionX := position;

						IF (side = 0) THEN
							position := position + 1000;
						ELSE
							position := position - 1000;
						END_IF;
					END_IF;

				ELSIF (Section[i].sectionType = SECTION_TYPE_N180) OR (Section[i].sectionType = SECTION_TYPE_W180L) THEN
					// Advance to next side when a curve follows straights,
					// or when a curve already exists on the current side.
					IF (side < 2) AND ((sideLength[side] > 0) OR (curveHSection[side] >= 0)) THEN
						side := side + 1;

						IF (side = 1) THEN
							modelIndex := 64 - sideLength[0];
							Data.CurvePositionX := position;
						END_IF;
					END_IF;

					IF (side = 1) THEN
						curveSide := 1;
					ELSE
						curveSide := 0;
					END_IF;

					IF (curveHSection[curveSide] < 0) THEN
						Section[i].side := curveSide;
						curveHSection[curveSide] := i;

						IF (Section[i].sectionType = SECTION_TYPE_N180) THEN
							Data.N180SectionVisible[curveSide] := TRUE;
						ELSE
							Data.W180SectionVisible[curveSide] := TRUE;
						END_IF;

						curveType := Section[i].sectionType;
					END_IF;

				ELSIF (Section[i].sectionType = SECTION_TYPE_W180R) THEN
					IF (side = 1) THEN
						curveSide := 1;
					ELSE
						curveSide := 0;
					END_IF;

					Section[i].side := curveSide;

				ELSE
					// unhandled section type

				END_IF;
			END_FOR;

			IF (curveType = SECTION_TYPE_N180) THEN
				Data.StraightSectionPositionY := 0;
				straightPalletPositionY[0] := -236;
				straightPalletPositionY[1] := 236;
			ELSE	// W180
				Data.StraightSectionPositionY := 365.5;
				straightPalletPositionY[0] := -236;
				straightPalletPositionY[1] := 600.5;
			END_IF;

			visuStep := visuSTEP_RUN;

		visuSTEP_RUN:
			// get actual pallet positions
			SuperTrakGetPalletInfo(ADR(Pallet), 128, FALSE);

			FOR i := 0 TO 127 DO
				IF (Pallet[i].section >= 1) AND (Pallet[i].section <= 99) THEN
					h := sectionLookup[ Pallet[i].section ];
				ELSE
					h := -1;
				END_IF;

				IF (h >= 0) THEN
					// display this pallet
					Data.Pallet[i].Visible := TRUE;
					position := DINT_TO_REAL(Pallet[i].position) / 1000;

					IF (Section[h].sectionType = SECTION_TYPE_1M) OR (Section[h].sectionType = SECTION_TYPE_1M_LP) THEN
						IF (Section[h].side = 0) THEN
							Data.Pallet[i].X := Section[h].positionX + position;
							Data.Pallet[i].Y := straightPalletPositionY[0];
							Data.Pallet[i].RZ := 0;
						ELSE
							Data.Pallet[i].X := Section[h].positionX - position;
							Data.Pallet[i].Y := straightPalletPositionY[1];
							Data.Pallet[i].RZ := 180;
						END_IF;

					ELSIF (Section[h].sectionType = SECTION_TYPE_N180) THEN
						// approximate the shape of the curve
						IF (position <= 15) THEN
							Data.Pallet[i].X := position;
							Data.Pallet[i].Y := -236;
							Data.Pallet[i].RZ := 0;
						ELSIF (position < 1015) THEN
							angle := brmPI * (position - 15) / 1000;
							Data.Pallet[i].X := 15 + (355 * SIN(angle)) - (15 * SIN(angle * 3));
							Data.Pallet[i].Y := (-257 * COS(angle)) + (21 * COS(angle * 3));
							Data.Pallet[i].RZ := 90 - 90 * COS(angle);
						ELSE
							Data.Pallet[i].X := 1030 - position;
							Data.Pallet[i].Y := 236;
							Data.Pallet[i].RZ := 180;
						END_IF;

						IF (Section[h].side = 0) THEN
							Data.Pallet[i].X := -Data.Pallet[i].X;
							Data.Pallet[i].Y := -Data.Pallet[i].Y;
							Data.Pallet[i].RZ := Data.Pallet[i].RZ - 180;
						ELSE
							Data.Pallet[i].X := Data.Pallet[i].X + Data.CurvePositionX;
						END_IF;

					ELSIF (Section[h].sectionType = SECTION_TYPE_W180L) THEN
						IF (position > 100) THEN
							angle := (position - 100) / W180_RADIUS * 180 / brmPI;
							position := 100;
						ELSE
							angle := 0;
						END_IF;

						IF (Section[h].side = 0) THEN
							Data.Pallet[i].X := -position - W180_RADIUS * SIN(angle * brmPI / 180);
							Data.Pallet[i].Y := 181.75 + W180_RADIUS * COS(angle * brmPI / 180);
							angle := angle + 180;
						ELSE
							Data.Pallet[i].X := position + Data.CurvePositionX + W180_RADIUS * SIN(angle * brmPI / 180);
							Data.Pallet[i].Y := 181.75 - W180_RADIUS * COS(angle * brmPI / 180);
						END_IF;

						Data.Pallet[i].RZ := angle;

					ELSIF (Section[h].sectionType = SECTION_TYPE_W180R) THEN
						IF (position > 650) THEN
							angle := 180;
							position := 759.347 - position;
						ELSE
							angle := (position / W180_RADIUS * 180 / brmPI) + 90;
							position := 100;
						END_IF;

						IF (Section[h].side = 0) THEN
							angle := angle + 180;
							Data.Pallet[i].X := -position - W180_RADIUS * ABS(SIN(angle * brmPI / 180));
							Data.Pallet[i].Y := 181.75 - W180_RADIUS * ABS(COS(angle * brmPI / 180));
						ELSE
							Data.Pallet[i].X := position + Data.CurvePositionX + W180_RADIUS * ABS(SIN(angle * brmPI / 180));
							Data.Pallet[i].Y := 181.75 + W180_RADIUS * ABS(COS(angle * brmPI / 180));
						END_IF;

						Data.Pallet[i].RZ := angle;

					END_IF;

				ELSE
					// hide this pallet
					Data.Pallet[i].Visible := FALSE;
					Data.Pallet[i].X := 0;
					Data.Pallet[i].Y := 0;
					Data.Pallet[i].RZ := 0;

				END_IF;
			END_FOR;

		ELSE
			// error or unhandled state; do nothing

	END_CASE;

END_PROGRAM
```

#### Types.typ - Local data types
```iecst
TYPE
	RoboVisuPallet_t : 	STRUCT
		Visible : BOOL; (*byte 0*)
		reserved_1 : USINT; (*byte 1*)
		Text : STRING[5]; (*Text / bytes 2-7*) (*STRING[n] = char[n + 1] = n characters plus terminator*)
		X : REAL; (*Position.X / bytes 8-11*)
		Y : REAL; (*Position.Y / bytes 12-15*)
		RZ : REAL; (*Orientation.RotZ / bytes 16-19*)
	END_STRUCT;
	RoboVisuData_t : 	STRUCT
		StraightSectionVisible : ARRAY[0..63]OF BOOL; (*bytes 0-63*)
		N180SectionVisible : ARRAY[0..1]OF BOOL; (*bytes 64-65*)
		W180SectionVisible : ARRAY[0..1]OF BOOL; (*bytes 66-67*)
		StraightSectionPositionY : REAL; (*bytes 68-71*)
		CurvePositionX : REAL; (*bytes 72-75*)
		reserved_76 : REAL; (*bytes 76-79*)
		reserved_80 : ARRAY[0..47]OF USINT; (*bytes 80-127*)
		reserved_128 : ARRAY[0..383]OF USINT; (*bytes 128-511*)
		Pallet : ARRAY[0..127]OF RoboVisuPallet_t; (*bytes 512-3071*)
	END_STRUCT;
	SectionInfo_t : 	STRUCT
		userAddress : UINT;
		sectionType : UINT;
		side : INT;
		modelIndex : INT;
		positionX : REAL;
	END_STRUCT;
END_TYPE
```

#### Variables.var - Local variables
```iecst
(*Visualization program states*)
VAR CONSTANT
	visuSTEP_INITIALIZE : USINT := 0;
	visuSTEP_GET_SECTION_COUNT : USINT := 1;
	visuSTEP_GET_SECTION_ADDRS : USINT := 2;
	visuSTEP_GET_SECTION_TYPES : USINT := 3;
	visuSTEP_SETUP_SECTIONS : USINT := 10;
	visuSTEP_RUN : USINT := 42;
	visuSTEP_ERROR : USINT := 99;
END_VAR
(*SuperTrak section types*)
VAR CONSTANT
	SECTION_TYPE_1M : UINT := 0;
	SECTION_TYPE_N180 : UINT := 1;
	SECTION_TYPE_1M_LP : UINT := 2;
	SECTION_TYPE_W180L : UINT := 3;
	SECTION_TYPE_W180R : UINT := 4;
END_VAR
(*Miscellaneous constants*)
VAR CONSTANT
	W180_RADIUS : REAL := 418.75;
END_VAR
(*Miscellaneous variables*)
VAR
	angle : REAL := 0.0;
	h : INT := 0;
	i : UINT := 0;
	position : REAL := 0.0;
	result : UINT := 0;
	visuStep : USINT := 0;
END_VAR
(*Visualization variables*)
VAR
	Data : RoboVisuData_t := (0); (*exported to Robotic Visualization*)
	sectionCount : UINT := 0;
	Section : ARRAY[0..63] OF SectionInfo_t; (*index = hSection*)
	Pallet : ARRAY[0..127] OF SuperTrakPalletInfo_t := [128(0)];
	sectionLookup : ARRAY[0..99] OF INT := [100(-1)]; (*index = user address, value = hSection*)
	straightPalletPositionY : ARRAY[0..1] OF REAL := [2(0.0)];
END_VAR
(*Setup variables*)
VAR
	curveHSection : ARRAY[0..1] OF INT := [2(-1)];
	curveSide : INT := 0;
	curveType : UINT := 0;
	modelIndex : INT := 0;
	side : INT := 0;
	sideLength : ARRAY[0..1] OF UINT := [2(0)];
END_VAR
(*SuperTrak service channel*)
VAR
	servChanResponseUINT : {REDUND_UNREPLICABLE} ARRAY[0..63] OF UINT;
END_VAR
```

### Package Logical/Source/Axis - Control the axis

### Program Logical/Source/Axis/AxisCtrl (IEC) - Control the axis

#### Main.st
```iecst
(*****************************************************************************
 * Copyright: COPYRIGHT (C) BERNECKER + RAINER, AUSTRIA
 *****************************************************************************
 * Author:  B+R  Created:  May 03, 2022/14:05 PM
 *****************************************************************************
 * Description: Implementation of the SDC-Axis
 ******************************************************************************)
PROGRAM _INIT

	// Initialize the function block
	gMpAxisBasic_0.Enable 				:= TRUE;
	gMpAxisBasic_0.MpLink 				:= ADR(gAxis1);
	gMpAxisBasic_0.Parameters			:= ADR(gMpAxisBasicParam);

	gMpAxisBasicParam.Velocity			:= 4000;
	gMpAxisBasicParam.Acceleration		:= 10000;
	gMpAxisBasicParam.Deceleration		:= 10000;
	gMpAxisBasicParam.Jog.Velocity		:= 1000;
	gMpAxisBasicParam.Jog.Acceleration	:= 10000;
	gMpAxisBasicParam.Jog.Deceleration	:= 10000;

	gMpAxisBasicParam.Jog.LimitPosition.FirstPosition := 500;
	gMpAxisBasicParam.Jog.LimitPosition.LastPosition := 3200;

END_PROGRAM

PROGRAM _CYCLIC
	// Home the axis if the SuperTrak-Sections is enabled
	IF gAllSectionsEnabled THEN
		gMpAxisBasic_0.Power 			:= TRUE;
	END_IF
	// Home the axis if its power on
	IF gMpAxisBasic_0.PowerOn AND NOT(gMpAxisBasic_0.IsHomed) THEN
		gMpAxisBasic_0.Home 			:= TRUE;
	END_IF
	// Reset the Input if the homing is done
	IF EDGEPOS(gMpAxisBasic_0.IsHomed) THEN
		gMpAxisBasic_0.Home				:= FALSE;
	END_IF

	//Call of the function block
	gMpAxisBasic_0();

END_PROGRAM

PROGRAM _EXIT

	gMpAxisBasic_0.Enable				:= FALSE;
	gMpAxisBasic_0();

END_PROGRAM
```

- Visualisation Logical/mappView (not shown)


Listed in the project but not available here: Logical/Global.typ, Logical/Source/SuperTrak/ST_Main/Types.typ
